{attribute 'no_explicit_call' := 'do not call this function block directly'} 
FUNCTION_BLOCK ABSTRACT Enumerator EXTENDS Object IMPLEMENTS IEnumerator
VAR
	_CurrentIndex : DINT := -1;
END_VAR

// Shows curent collection element
PROPERTY ABSTRACT Current : PVOID
GET
END_GET
END_PROPERTY

{attribute "object_name" := "MoveNext"}
// Moves Current pointer to next collection element
METHOD ABSTRACT MoveNext : BOOL
END_METHOD

{attribute "object_name" := "Reset"}
// Sets the enumerator to its initial position, which is before the first element in the collection
METHOD Reset
_CurrentIndex := -1;
END_METHOD

END_FUNCTION_BLOCK

(* stored: Version 1.1.0.1
   POU Enumerator: Id {1ba2dded-f68b-058f-2c2a-52c4eba159dc}, SpecialFunc None
   Property Current: Id {ee0b79eb-0bf9-0862-23fc-a4125a07061d}
   Get Get: Id {3a2ce99c-cf70-0aca-02a4-2206750aa89d}
   Method MoveNext: Id {a7e98f26-ff1f-0da4-0d33-c119f7486eaa}
   Method Reset: Id {cf4a0ab3-611e-0cee-0831-cedc404a7abd} *)
